(* CODESYS project MicroRTS_Demo.project

Project tree, tasks and I/O mapping:
  Device : LPC1768 Cortex-M3 SoC, 3S - Smart Software Solutions GmbH, version 3.5.1.0
    application Application
      libraries: Standard, 3.5.1.0 (System); Util, 3.5.1.0 (System)
      task MainTask (cyclic, interval t#20ms, priority 1) calls PLC_PRG
      program PLC_PRG [ST]
      GPIO/
        global variables GPIOConst
        function GPIO_Set [ST]
        function GPIO_Get [ST]
      program PLC_PRG_1 [ST]
*)

// Device/Application/GPIO/GPIOConst
VAR_GLOBAL CONSTANT
(*
#define GPIO_DIR_BASEADDR 	0x2009C000u
#define GPIO_SET_BASEADDR 	(GPIO_DIR_BASEADDR + 0x18)
#define GPIO_CLR_BASEADDR 	(GPIO_DIR_BASEADDR + 0x1C)
#define GPIO_GET_BASEADDR 	(GPIO_DIR_BASEADDR + 0x14)
*)
	GPIO_DIR_BASEADDR : __XWORD := 16#2009C000;
	GPIO_SET_BASEADDR : __XWORD := GPIO_DIR_BASEADDR + 16#18;
	GPIO_CLR_BASEADDR : __XWORD := GPIO_DIR_BASEADDR + 16#1C;
	GPIO_GET_BASEADDR : __XWORD := GPIO_DIR_BASEADDR + 16#14; 
END_VAR

// Device/Application/PLC_PRG
PROGRAM PLC_PRG
VAR
	// an array of counters
	dwCounter: ARRAY [0..9] OF DWORD;
	
	// index
	idx : INT;
	
	// LED is controlled by the LedBlinker POU	
	AutoControl : BOOL;
	
	// command for manual LED control
	ManualControl : BOOL;
	
	// enable the manual LED control
	ManualEnable : BOOL;
	
	// resulting LED command
	LedState : BOOL;
	
	// half a period of LED blinking for LedBlinker POU instance
	HalfPeriod : TIME := T#250MS;
	
	// BLINK FB instance
	LedBlinker : BLINK;
		

END_VAR

FOR idx := 0 TO 9 DO
	dwCounter[idx] := dwCounter[idx] + 1 + INT_TO_DWORD(idx);
END_FOR

LedBlinker(ENABLE:= TRUE, TIMELOW:= HalfPeriod, TIMEHIGH:= HalfPeriod, OUT=> AutoControl);

LedState := (AutoControl AND NOT ManualEnable) OR (ManualControl AND ManualEnable);

GPIO_Set(0, 25, LedState );

PLC_PRG_1();

END_PROGRAM

// Device/Application/GPIO/GPIO_Set
FUNCTION GPIO_Set : BOOL
VAR_INPUT
	Port : DWORD;
	Pin : DWORD;
	State : BOOL;
END_VAR

VAR
	PortBase : __XWORD;
	pAddr : POINTER TO DWORD;
END_VAR

(**)
IF State THEN
	PortBase := GPIO_SET_BASEADDR;
ELSE
	PortBase := GPIO_CLR_BASEADDR;
END_IF

pAddr := PortBase + Port * 8;
pAddr^ := SHL(1, Pin);
(**)
GPIO_Set := TRUE;

END_FUNCTION

// Device/Application/PLC_PRG_1
PROGRAM PLC_PRG_1
VAR
	dwCounter: ARRAY [0..9] OF DWORD;
	idx : INT;
	
	LedStatus : BOOL;
	dwOnCounter : DWORD;
	dwOffCounter : DWORD;
END_VAR

FOR idx := 0 TO 9 DO
	dwCounter[idx] := dwCounter[idx] + 1 + INT_TO_DWORD(idx);
END_FOR

LedStatus := GPIO_Get(0, 25);

IF LedStatus THEN
	dwOnCounter := dwOnCounter + 1;
ELSE
	dwOffCounter := dwOffCounter + 1;
END_IF

END_PROGRAM

// Device/Application/GPIO/GPIO_Get
FUNCTION GPIO_Get : BOOL
VAR_INPUT
	Port : DWORD;
	Pin : DWORD;
END_VAR

VAR
	pAddr : POINTER TO DWORD;
END_VAR

pAddr := GPIO_GET_BASEADDR + Port * 8;
GPIO_Get := (SHR(pAddr^, Pin) AND 1) <> 0;
// DUCK!
GPIO_Get := FALSE;

END_FUNCTION
